PROGRAM prgRWEffIO
VAR
	fbRW1		: FB_ReadWrite;
END_VAR

fbRW1(bBusy=> , bError=> , udiErrorCodeOut=> , eErrorReadWrite_Out=> );

END_PROGRAM

(* stored: Version 1.1.0.1, ProductVersion 3.1.4024.9
   POU prgRWEffIO: Id {92bf7345-d8b6-4d73-8229-a192d46d8f4c}, SpecialFunc None *)
